// TIA Portal V21 program export: 7 tag tables, 1 data types, 2 data blocks, 11 code blocks (in call order from the OBs), 0 instance data blocks

VAR_GLOBAL   // PLC tag table "INSTRUMENTOS_ALARMES (ETA)"
   "NIVEL_MUITO_ALTO (ETA)" AT %M60.0 : Bool;
   "PRESSAO_ALTA (ETA)" AT %M60.1 : Bool;
END_VAR

VAR_GLOBAL   // PLC tag table "INSTRUMENTOS (ETA)"
   "FIT-01_STS" AT %M61.0 : Bool;
   "LIT-01_STS" AT %M61.1 : Bool;
END_VAR

VAR_GLOBAL   // PLC tag table "LadderTags"
   Start AT %M26.0 : Bool;
   Stop AT %M26.1 : Bool;
   Cmd_Motor1 AT %M26.2 : Bool;
   Falha_M1 AT %M26.3 : Bool;
   Nivel_Alto AT %M26.4 : Bool;
   Auto AT %M26.5 : Bool;
   Alarme AT %M26.6 : Bool;
   Reset AT %M26.7 : Bool;
   Manutencao AT %M27.0 : Bool;
   Pronto AT %M27.1 : Bool;
   Sensor_Falha AT %M27.2 : Bool;
   Temp_OK AT %M27.3 : Bool;
   Temperatura AT %MW28 : Int;
   Setpoint AT %MW30 : Int;
END_VAR

VAR_GLOBAL   // PLC tag table "SmokeTags"
   Smoke_Bit AT %M10.0 : Bool;
   Smoke_Out AT %M10.1 : Bool;
   Smoke_Int AT %MW12 : Int;
END_VAR

VAR_GLOBAL   // PLC tag table "PARTIDAS (ETA)"
   "ETA-P01_FALHA" AT %M60.2 : Bool;
END_VAR

VAR_GLOBAL   // PLC tag table "SOPRADOR_DESARENADOR (S-01A)"
   "S-01A_RESERVA_01" AT %M5512.0 : Bool;
   "S-01A_RESERVA_02" AT %M5512.1 : Bool;
   "S-01A_RESERVA_DINT_01" AT %MD5513 : DInt;
   "S-01A_STS_HABILITA_IMPAR_&" AT %M5506.4 : Bool;   // Status: Condições para partida do equipamento S-01A estão OK
   "S-01A_FALHA" AT %M5500.7 : Bool;   // Status: Falha geral do equipamento S-01A
   "S-01A_STS_FALHA_NAO_LIGOU" AT %M5506.1 : Bool;   // Status: Falha de partida do equipamento S-01A
   "S-01A_CMD_HABILITA_LIGA_AUTO2" AT %M5500.2 : Bool;   // Comando: Habilitação para partida em modo automático para o equipamento S-01A
   "S-01A_SP_SETPOINT_AUTO" AT %MW5502 : Int;   // Setpoint: Valor de referência em modo automático para o equipamento S-01A
   "S-01A_STS_HABILITA_PAR_&" AT %M5506.5 : Bool;   // Status: Condições para partida do equipamento S-01A estão OK
   "S-01A_CMD_BOTAO_RESET_FALHA" AT %M5500.0 : Bool;   // Comando: Botão de reset de falhas para o equipamento S-01A
   "S-01A_STS_VAR_MONITORADA" AT %MD5508 : Real;   // Status: Variável monitorada (Ex: vibração, temperatura) do equipamento S-01A
   "S-01A_STS_REMOTO_AUTO" AT %M5507.3 : Bool;   // Status: Comando Remoto em modo Automático para o equipamento S-01A
   "S-01A_STS_REMOTO_MANUAL" AT %M5507.4 : Bool;   // Status: Comando Remoto em modo Manual para o equipamento S-01A
   "S-01A_STS_LIGADO_PROFINET" AT %M5506.6 : Bool;   // Status: Comunicação Profinet OK com o equipamento S-01A
   "S-01A_STS_ALTERNANCIA_OK" AT %M5506.0 : Bool;   // Tag de controle/status/falha para o equipamento S-01A
   "S-01A_CMD_RESET_LIGA" AT %M5500.6 : Bool;   // Comando: Reset do comando Ligar o equipamento S-01A
   "S-01A_CMD_RESET_FALHA_PROFINET" AT %M5500.5 : Bool;   // Comando: Reset de falha Profinet para o equipamento S-01A
   "S-01A_STS_MODO_REMOTO" AT %M5507.2 : Bool;   // Status: Chave seletora do equipamento S-01A em Remoto
   "S-01A_LIGADO" AT %M5501.0 : Bool;   // Status: Equipamento S-01A em operação
   "S-01A_CMD_HABILITA_LIGA_AUTO" AT %M5500.1 : Bool;   // Comando: Habilitação para partida em modo automático para o equipamento S-01A
   "S-01A_STS_LOCAL_MANUAL" AT %M5507.0 : Bool;   // Status: Comando Local em modo Manual para o equipamento S-01A
   "S-01A_STS_FALHA_PROFINET" AT %M5506.2 : Bool;   // Status: Falha de comunicação Profinet com o equipamento S-01A
   "S-01A_STS_SUCCAO_OK" AT %M5507.5 : Bool;   // Status: Condição de sucção OK para a bomba S-01A
   "S-01A_STS_MODO_LOCAL" AT %M5507.1 : Bool;   // Status: Chave seletora do equipamento S-01A em Local
   "S-01A_STS_HABILITA" AT %M5506.3 : Bool;   // Status: Condições para partida do equipamento S-01A estão OK
   "S-01A_STS_LOCAL_AUTO" AT %M5506.7 : Bool;   // Status: Comando Local em modo Automático para o equipamento S-01A
   "S-01A_CMD_LIGA_PROFINET" AT %M5500.4 : Bool;   // Comando: Partida via Profinet para o equipamento S-01A
   "S-01A_SP_SETPOINT_MANUAL" AT %MW5504 : Int;   // Setpoint: Valor de referência em modo manual para o equipamento S-01A
   "S-01A_CMD_LIGA_BOMBA" AT %M5500.3 : Bool;   // Comando: Ligar/Partir a bomba S-01A
END_VAR

VAR_GLOBAL   // PLC tag table "BOMBA (BH-01B)"
END_VAR

TYPE "MotorDados"
VERSION : 0.1
   STRUCT
      Liga : Bool;
      Ligado : Bool;
      Numero : Int;
   END_STRUCT;
END_TYPE

DATA_BLOCK "DB GLOBAL"
{ S7_Optimized_Access := 'TRUE' }
VERSION : 0.1
   STRUCT
      "Motor_BH-01A" : "MotorDados";
      "Motor_BH-01B" : "MotorDados";
   END_STRUCT;

BEGIN
END_DATA_BLOCK

DATA_BLOCK "ALARMES_MODULOS"
{ S7_Optimized_Access := 'TRUE' }
VERSION : 0.1
   STRUCT
      "QA-01" : STRUCT
         WORD_1 : Word;
         WORD_2 : Word;
      END_STRUCT;
   END_STRUCT;

BEGIN
END_DATA_BLOCK

DATA_BLOCK "DB INSTRUMENTOS"
{ S7_Optimized_Access := 'TRUE' }
VERSION : 0.1
   STRUCT
      ETA : STRUCT
         "FIT-01" : STRUCT
            WORD_STS : Word;
            CMD_AF : Int;
            CMD_LIM : Int;
         END_STRUCT;
         "LIT-01" : STRUCT
            WORD_STS : Word;
            CMD_AF : Int;
            CMD_LIM : Int;
         END_STRUCT;
      END_STRUCT;
   END_STRUCT;

BEGIN
END_DATA_BLOCK

DATA_BLOCK "DB_BITS_TO_WORD_FIT-01"
{ S7_Optimized_Access := 'TRUE' }
VERSION : 0.1
"FB BITS TO WORD"

BEGIN
END_DATA_BLOCK

ORGANIZATION_BLOCK "OB_MOLDE_ALARMES"   // OB1, LAD, ProgramCycle
TITLE = "Main Program Sweep (Cycle)"
{ S7_Optimized_Access := 'TRUE' }
VERSION : 0.1
// stored: AutoNumber true, IsIECCheckEnabled false, SetENOAutomatically false
   VAR_INPUT
      Initial_Call : Bool;   // Initial call of this OB
      Remanence : Bool;   // =True, if remanent data are available
   END_VAR
BEGIN

REGION Network 1: FC Alarmes: Paineis
   // comentário da chamada da fc 1
END_REGION
END_ORGANIZATION_BLOCK

ORGANIZATION_BLOCK "MODULE_ERROR_MOLDE"   // OB123, LAD, ProgramCycle
TITLE = MODULE_ERROR_MOLDE
{ S7_Optimized_Access := 'TRUE' }
VERSION : 0.1
// stored: AutoNumber true, IsIECCheckEnabled false, SetENOAutomatically false
   VAR_INPUT
      Initial_Call : Bool;
      Remanence : Bool;
   END_VAR
BEGIN

REGION Network 1: Molde: falha modulo HW 999
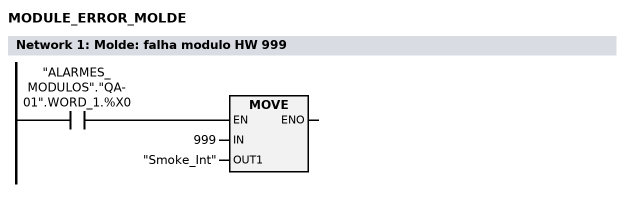
   RUNG wire#powerrail
      Contact( "ALARMES_MODULOS"."QA-01".WORD_1.%X0 )
      { S7_GenerateENO := "TRUE" } Move(in := 999, out1 := "Smoke_Int")
   END_RUNG
   // the same network as SCL:
   IF "ALARMES_MODULOS"."QA-01".WORD_1.%X0 THEN <??.?> := 999; END_IF;
END_REGION
END_ORGANIZATION_BLOCK

ORGANIZATION_BLOCK "OB_INSTRUMENTOS"   // OB130, LAD, ProgramCycle
TITLE = OB_INSTRUMENTOS
{ S7_Optimized_Access := 'TRUE' }
VERSION : 0.1
// stored: AutoNumber true, IsIECCheckEnabled false, SetENOAutomatically false
   VAR_INPUT
      Initial_Call : Bool;
      Remanence : Bool;
   END_VAR
BEGIN
END_ORGANIZATION_BLOCK

FUNCTION "PARTIDA_SOPRADOR_1 (S-01A)" : Void   // FC148, LAD
{ S7_Optimized_Access := 'TRUE' }
VERSION : 0.1
// Network 1: Set memórias entradas digitais
// Network 2: Function Block FALHA
// Network 3: MODO AUTOMÁTICO: Condições para Modo Automático
// Network 4: Alternância/Rotatividade de bombas Principal-Reserva
// Network 5: Function Block CONDIÇÃO DE PARTIDA
// Network 6: Setpoint Manual - Velocidade Proporcial ao Sinal de Saída
// Network 7: Reset Comando Liga
// Network 8: Intertravamento para habilitar o botão liga na IHM
// Network 9: Intertravamento de Segurança
// Network 10: Bloco de Controle Inversor Profinet
// Network 11: Aciona saída digital para partir o motor/bomba
// Network 1: Set memórias entradas digitais
// Network 2: Function Block FALHA
// Network 3: MODO AUTOMÁTICO: Condições para Modo Automático
// Network 4: Alternância/Rotatividade de bombas Principal-Reserva
// Network 5: Function Block CONDIÇÃO DE PARTIDA
// Network 6: Reset Comando Liga
// Network 7: Function Block MODOS DE OPERAÇÃO - Atribuição dos Modos de Operação
// Network 8: Intertravamento para habilitar o botão liga na IHM
// Network 9: Intertravamento de Segurança
// Network 10: Function Block SUCÇÃO OK
// Network 11: Aciona saída digital para partir o motor/bomba
// Network 12: Function Block HORÍMETRO - Tempo de bomba ligada em horas
// stored: AutoNumber true, IsIECCheckEnabled false, SetENOAutomatically false, UDAEnableTagReadback false
   VAR_TEMP   // added for the SCL form of the ladder/FBD networks
      _w1 : Bool;
   END_VAR
BEGIN

REGION Network 1: Set memórias entradas digitais
   // Instanciando entradas digitais em PLC Tags "%M " Address
   // 
   // MODO LOCAL: Indica Operação Local da bomba.
   // MODO REMOTO: Indica Operação Remoto da bomba (IHM).
   // LIGADO: Indica bomba ligada (caso, via sinal discreto).
   // FALHA: Sinal de Falha (caso, via sinal discreto).
   // Instanciando entradas digitais em PLC Tags "M" Address
   // 
   // MODO LOCAL: Indica Operação Local da bomba
   // MODO REMOTO: Indica Operação Remoto da bomba (IHM)
   // LIGADO: Indica bomba ligada
   // FALHA: Sinal de Falha
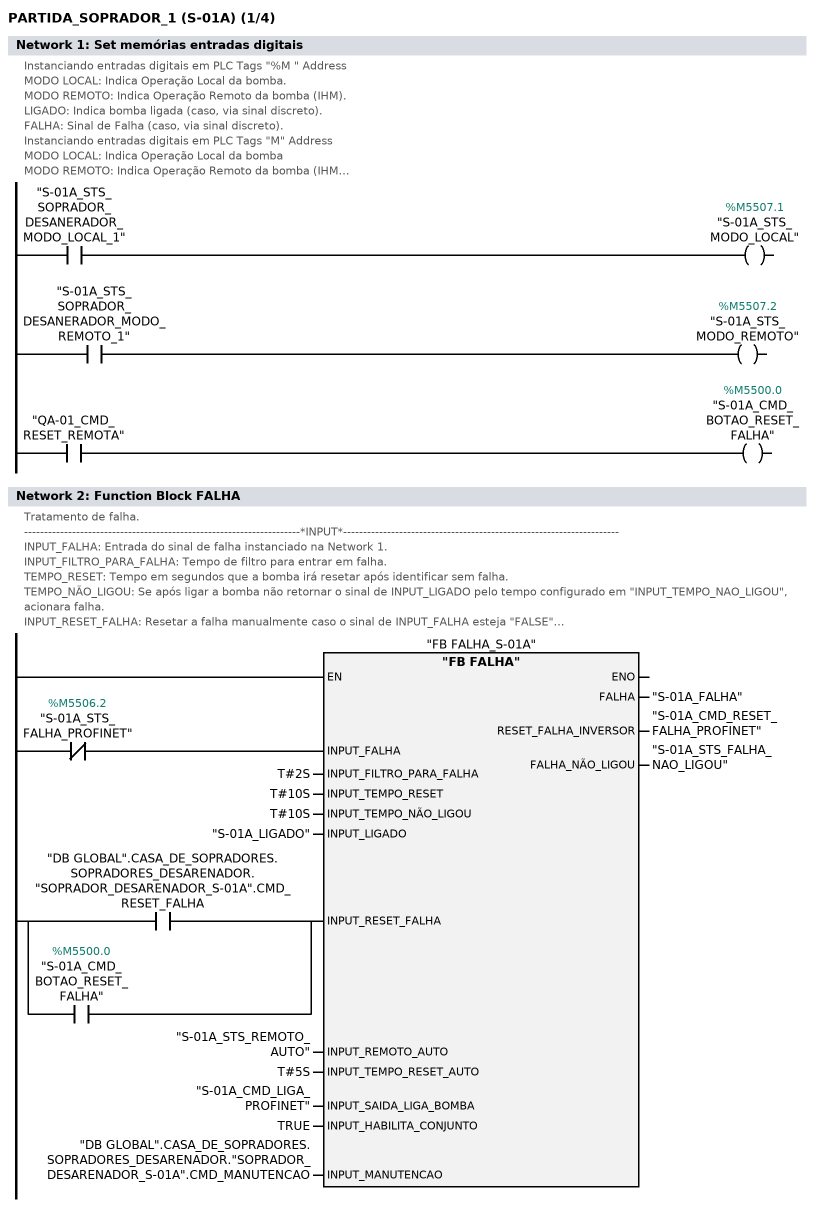
   RUNG wire#powerrail
      Contact( "S-01A_STS_SOPRADOR_DESANERADOR_MODO_LOCAL_1" )
      Coil( "S-01A_STS_MODO_LOCAL" )
   END_RUNG
   RUNG wire#powerrail
      Contact( "S-01A_STS_SOPRADOR_DESANERADOR_MODO_REMOTO_1" )
      Coil( "S-01A_STS_MODO_REMOTO" )
   END_RUNG
   RUNG wire#powerrail
      Contact( "QA-01_CMD_RESET_REMOTA" )
      Coil( "S-01A_CMD_BOTAO_RESET_FALHA" )
   END_RUNG
   // the same network as SCL:
   "S-01A_STS_MODO_LOCAL" := "S-01A_STS_SOPRADOR_DESANERADOR_MODO_LOCAL_1";
   "S-01A_STS_MODO_REMOTO" := "S-01A_STS_SOPRADOR_DESANERADOR_MODO_REMOTO_1";
   "S-01A_CMD_BOTAO_RESET_FALHA" := "QA-01_CMD_RESET_REMOTA";
END_REGION

REGION Network 2: Function Block FALHA
   // Tratamento de falha.
   // ---------------------------------------------------------------------*INPUT*---------------------------------------------------------------------
   // INPUT_FALHA: Entrada do sinal de falha instanciado na Network 1.
   // INPUT_FILTRO_PARA_FALHA: Tempo de filtro para entrar em falha.
   // TEMPO_RESET: Tempo em segundos que a bomba irá resetar após identificar sem falha.
   // TEMPO_NÃO_LIGOU: Se após ligar a bomba não retornar o sinal de INPUT_LIGADO pelo tempo configurado em "INPUT_TEMPO_NAO_LIGOU", acionara falha.
   // INPUT_RESET_FALHA: Resetar a falha manualmente caso o sinal de INPUT_FALHA esteja "FALSE".
   // INPUT_REMOTO_AUTO: Caso o equipamento entrar em estado de "FALHA" em "REMOTO_AUTOMATICO" o bloco fará um reset com atraso pelo tempo "INPUT_TEMPO_RESET_AUTO".
   // INPUT_TEMPO_RESET_AUTO: Caso em "REMOTO_AUTO", para resetar será contado o tempo de entrada.
   // INPUT_SAIDA_LIGA_BOMBA: Comando de saída para acionar o equipamento.
   // INPUT_HABILITA_CONJUNTO: Comando para casos de Principal e Reserva (padrão "TRUE").
   // INPUT_MANUTENCAO: Comando de manutenção do equipamento intertrava qualquer acionamento e status de "FALHA".
   // ---------------------------------------------------------------------*OUTPUT*---------------------------------------------------------------------
   // FALHA: Sinal de saída de "FALHA" do equipamento.
   // RESET_FALHA_INVERSOR: Comando enviado para reset do inversor em caso de "FALHA".
   // FALHA_NAO_LIGOU: Caso esteja sendo enviado o comando para "LIGAR" e não receber o feedback de ligado, no tempo de "TEMPO_NÃO_LIGOU", o equiapamento entra em "FALHA".
   // Tratamento de falha da bomba
   // INPUT_FALHA: Entrada do sinal de falha instanciado na Network 1.
   // TEMPO_RESET: Tempo em segundos que a bomba irá resetar após identificar sem falha.
   // TEMPO_NÃO_LIGOU: Se após ligar a bomba não retornar o sinal de LIGADO pelo tempo configurado, acionara falha.
   // INPUT_RESET_FALHA: Resetar a falha manualmente caso o sinal de INPUT_FALHA esteja FALSE
   RUNG wire#powerrail
      "FB FALHA_S-01A"(INPUT_FALHA := wire#w1, INPUT_RESET_FALHA := wire#w2, INPUT_FILTRO_PARA_FALHA := T#2S, INPUT_TEMPO_RESET := T#10S, INPUT_TEMPO_NÃO_LIGOU := T#10S, INPUT_LIGADO := "S-01A_LIGADO", INPUT_REMOTO_AUTO := "S-01A_STS_REMOTO_AUTO", INPUT_TEMPO_RESET_AUTO := T#5S, INPUT_SAIDA_LIGA_BOMBA := "S-01A_CMD_LIGA_PROFINET", INPUT_HABILITA_CONJUNTO := TRUE, INPUT_MANUTENCAO := "DB GLOBAL".CASA_DE_SOPRADORES.SOPRADORES_DESARENADOR."SOPRADOR_DESARENADOR_S-01A".CMD_MANUTENCAO, FALHA => "S-01A_FALHA", RESET_FALHA_INVERSOR => "S-01A_CMD_RESET_FALHA_PROFINET", FALHA_NÃO_LIGOU => "S-01A_STS_FALHA_NAO_LIGOU")
   END_RUNG
   RUNG wire#powerrail
      I_Contact( "S-01A_STS_FALHA_PROFINET" )
   END_RUNG wire#w1
   RUNG wire#powerrail
      Contact( "DB GLOBAL".CASA_DE_SOPRADORES.SOPRADORES_DESARENADOR."SOPRADOR_DESARENADOR_S-01A".CMD_RESET_FALHA )
   END_RUNG wire#w2
   RUNG wire#powerrail
      Contact( "S-01A_CMD_BOTAO_RESET_FALHA" )
   END_RUNG wire#w2
   // the same network as SCL:
   "FB FALHA_S-01A"(INPUT_FALHA := NOT "S-01A_STS_FALHA_PROFINET",   // "FB FALHA"
                    INPUT_FILTRO_PARA_FALHA := T#2S,
                    INPUT_TEMPO_RESET := T#10S,
                    INPUT_TEMPO_NÃO_LIGOU := T#10S,
                    INPUT_LIGADO := "S-01A_LIGADO",
                    INPUT_RESET_FALHA := "DB GLOBAL".CASA_DE_SOPRADORES.SOPRADORES_DESARENADOR."SOPRADOR_DESARENADOR_S-01A".CMD_RESET_FALHA OR "S-01A_CMD_BOTAO_RESET_FALHA",
                    INPUT_REMOTO_AUTO := "S-01A_STS_REMOTO_AUTO",
                    INPUT_TEMPO_RESET_AUTO := T#5S,
                    INPUT_SAIDA_LIGA_BOMBA := "S-01A_CMD_LIGA_PROFINET",
                    INPUT_HABILITA_CONJUNTO := TRUE,
                    INPUT_MANUTENCAO := "DB GLOBAL".CASA_DE_SOPRADORES.SOPRADORES_DESARENADOR."SOPRADOR_DESARENADOR_S-01A".CMD_MANUTENCAO,
                    FALHA => "S-01A_FALHA",
                    RESET_FALHA_INVERSOR => "S-01A_CMD_RESET_FALHA_PROFINET",
                    FALHA_NÃO_LIGOU => "S-01A_STS_FALHA_NAO_LIGOU");
END_REGION

REGION Network 3: MODO AUTOMÁTICO: Condições para Modo Automático
   // ----------------------------------------------------------------------*INPUT*---------------------------------------------------------------------
   // ---------------------------------------------------------------------*OUTPUT*------------------------------------------------------------------
END_REGION

REGION Network 4: Alternância/Rotatividade de bombas Principal-Reserva
   // ----------------------------------------------------------------------*INPUT*---------------------------------------------------------------------
   // ---------------------------------------------------------------------*OUTPUT*------------------------------------------------------------------
END_REGION

REGION Network 5: Function Block CONDIÇÃO DE PARTIDA
   // Varredura de condicionais para ligar
   // ----------------------------------------------------------------------*INPUT*---------------------------------------------------------------------
   // INPUT_LIGADO: Entrada do sinal de ligado instanciado na Network 1.
   // INPUT_DESLIGADO: Entrada do sinal discreto "DESLIGADO" (caso, feedback via sinal discreto).
   // INPUT_FALHA: Entrada do sinal de falha da saída do bloco na Network 2.
   // INPUT_LOCAL: Entrada do sinal de modo local instanciado na Network 1.
   // INPUT_LOC_AUTO: Entrada do sinal do modo Local Automático
   // INPUT_REMOTO: Entrada do sinal de modo remoto instanciado na Network 1.
   // INPUT_FALHA_PROFNET: Entrada do sinal de Falha na comunicação Profinet.
   // INPUT_HABILITA_AUTO: Entrada do Sinal que habilita o modo Automático.
   // INPUT_CMD_LIGA: Entrada do sinal para acionar o equipamento.
   // CMD_MANUTENÇÃO:Comando de manutenção do equipamento intertrava qualquer acionamento.
   // CMD_MODO_OPERAÇÃO: Seleção do modo de operação do equipamento.
   // CMD_RESET_HORIMETRO: Comando para resetar o contador de Horas Trabalhadas.
   // 
   // 
   // ---------------------------------------------------------------------*OUTPUT*------------------------------------------------------------------
   // LIGA_BOMBA: Se TRUE, as condições estão OK para ligar na Network 11.
   // STATUS_MOTOR: Status de saída; 0 = DESLIGADO; 1 = LIGADO; 2 = FALHA; 3 = MANUTENÇÃO.
   // OUTPUT_REMOTO_AUTO: Saída indica que o motor/bomba está em modo Remoto Automático.
   // OUTPUT_MODO_OPERAÇÃO: Modo de operação local/remoto, manual/automático do equipamento
   // STS_HORIMETRO: Contabilização do tempo do equipamento em operação.
   // RESET_CMD_LIGA: Reset da memória de comando "LIGA" em casos do equipamento estar em modo "REMOTO_AUTOMATICO" ou "FALHA" ou "MANUTENÇÃO".
   // Varredura de condicionais para ligar
   // INPUT_LIGADO: Entrada do sinal de ligado instanciado na Network 1.
   // INPUT_FALHA: Entrada do sinal de falha da saída do bloco na Network 2.
   // INPUT_LOCAL: Entrada do sinal de modo local instanciado na Network 1.
   // INPUT_LOC_AUTO: Entrada do sinal do modo Local Automático
   // INPUT_REMOTO: Entrada do sinal de modo remoto instanciado na Network 1.
   // PARÂMETRO: Parâmetro de monitoramento para ligar e desligar a bomba em automático.
   // PARÂMETRO_LIGA/DESLIGA: Cadastros de programação liga/desliga em relação ao parâmetro.
   // CMD: Comandos recebidos pelo bloco
   // STATUS_MOTOR: Status de saída; 0 = DESLIGADO; 1 = LIGADO; 2 = FALHA; 3 = MANUTENÇÃO.
   // LIGA_BOMBA: Se TRUE, as condições estão OK para ligar na 5.
   // REMOTO_MAN: Saída indica que o motor/bomba está em modo Remoto Manual
   // REMOTO_AUTO: Saída indica que o motor/bomba está em modo Remoto Automático
   // LOCAL_MAN: Saída indica que o motor/bomba está em modo Local Manual
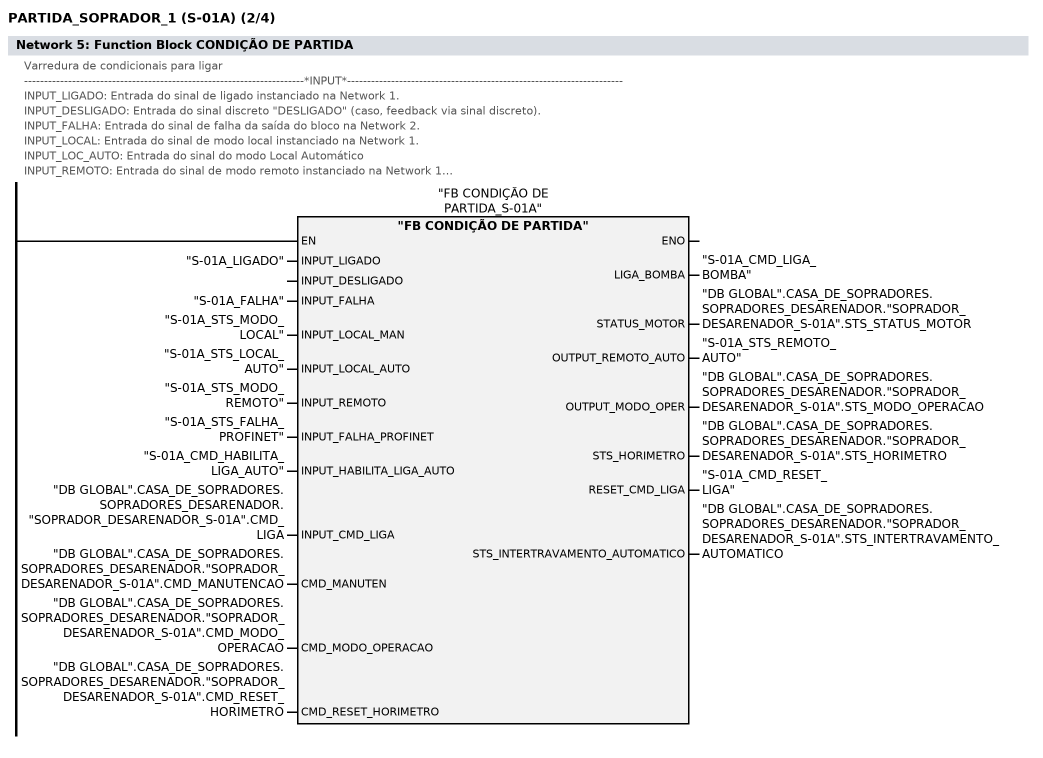
   RUNG wire#powerrail
      "FB CONDIÇÃO DE PARTIDA_S-01A"(INPUT_LIGADO := "S-01A_LIGADO", INPUT_DESLIGADO :=, INPUT_FALHA := "S-01A_FALHA", INPUT_LOCAL_MAN := "S-01A_STS_MODO_LOCAL", INPUT_LOCAL_AUTO := "S-01A_STS_LOCAL_AUTO", INPUT_REMOTO := "S-01A_STS_MODO_REMOTO", INPUT_FALHA_PROFINET := "S-01A_STS_FALHA_PROFINET", INPUT_HABILITA_LIGA_AUTO := "S-01A_CMD_HABILITA_LIGA_AUTO", INPUT_CMD_LIGA := "DB GLOBAL".CASA_DE_SOPRADORES.SOPRADORES_DESARENADOR."SOPRADOR_DESARENADOR_S-01A".CMD_LIGA, CMD_MANUTEN := "DB GLOBAL".CASA_DE_SOPRADORES.SOPRADORES_DESARENADOR."SOPRADOR_DESARENADOR_S-01A".CMD_MANUTENCAO, CMD_MODO_OPERACAO := "DB GLOBAL".CASA_DE_SOPRADORES.SOPRADORES_DESARENADOR."SOPRADOR_DESARENADOR_S-01A".CMD_MODO_OPERACAO, CMD_RESET_HORIMETRO := "DB GLOBAL".CASA_DE_SOPRADORES.SOPRADORES_DESARENADOR."SOPRADOR_DESARENADOR_S-01A".CMD_RESET_HORIMETRO, LIGA_BOMBA => "S-01A_CMD_LIGA_BOMBA", STATUS_MOTOR => "DB GLOBAL".CASA_DE_SOPRADORES.SOPRADORES_DESARENADOR."SOPRADOR_DESARENADOR_S-01A".STS_STATUS_MOTOR, OUTPUT_REMOTO_AUTO => "S-01A_STS_REMOTO_AUTO", OUTPUT_MODO_OPER => "DB GLOBAL".CASA_DE_SOPRADORES.SOPRADORES_DESARENADOR."SOPRADOR_DESARENADOR_S-01A".STS_MODO_OPERACAO, STS_HORIMETRO => "DB GLOBAL".CASA_DE_SOPRADORES.SOPRADORES_DESARENADOR."SOPRADOR_DESARENADOR_S-01A".STS_HORIMETRO, RESET_CMD_LIGA => "S-01A_CMD_RESET_LIGA", STS_INTERTRAVAMENTO_AUTOMATICO => "DB GLOBAL".CASA_DE_SOPRADORES.SOPRADORES_DESARENADOR."SOPRADOR_DESARENADOR_S-01A".STS_INTERTRAVAMENTO_AUTOMATICO)
   END_RUNG
   // the same network as SCL:
   "FB CONDIÇÃO DE PARTIDA_S-01A"(INPUT_LIGADO := "S-01A_LIGADO",   // "FB CONDIÇÃO DE PARTIDA"
                           INPUT_FALHA := "S-01A_FALHA",
                           INPUT_LOCAL_MAN := "S-01A_STS_MODO_LOCAL",
                           INPUT_LOCAL_AUTO := "S-01A_STS_LOCAL_AUTO",
                           INPUT_REMOTO := "S-01A_STS_MODO_REMOTO",
                           INPUT_FALHA_PROFINET := "S-01A_STS_FALHA_PROFINET",
                           INPUT_HABILITA_LIGA_AUTO := "S-01A_CMD_HABILITA_LIGA_AUTO",
                           INPUT_CMD_LIGA := "DB GLOBAL".CASA_DE_SOPRADORES.SOPRADORES_DESARENADOR."SOPRADOR_DESARENADOR_S-01A".CMD_LIGA,
                           CMD_MANUTEN := "DB GLOBAL".CASA_DE_SOPRADORES.SOPRADORES_DESARENADOR."SOPRADOR_DESARENADOR_S-01A".CMD_MANUTENCAO,
                           CMD_MODO_OPERACAO := "DB GLOBAL".CASA_DE_SOPRADORES.SOPRADORES_DESARENADOR."SOPRADOR_DESARENADOR_S-01A".CMD_MODO_OPERACAO,
                           CMD_RESET_HORIMETRO := "DB GLOBAL".CASA_DE_SOPRADORES.SOPRADORES_DESARENADOR."SOPRADOR_DESARENADOR_S-01A".CMD_RESET_HORIMETRO,
                           LIGA_BOMBA => "S-01A_CMD_LIGA_BOMBA",
                           STATUS_MOTOR => "DB GLOBAL".CASA_DE_SOPRADORES.SOPRADORES_DESARENADOR."SOPRADOR_DESARENADOR_S-01A".STS_STATUS_MOTOR,
                           OUTPUT_REMOTO_AUTO => "S-01A_STS_REMOTO_AUTO",
                           OUTPUT_MODO_OPER => "DB GLOBAL".CASA_DE_SOPRADORES.SOPRADORES_DESARENADOR."SOPRADOR_DESARENADOR_S-01A".STS_MODO_OPERACAO,
                           STS_HORIMETRO => "DB GLOBAL".CASA_DE_SOPRADORES.SOPRADORES_DESARENADOR."SOPRADOR_DESARENADOR_S-01A".STS_HORIMETRO,
                           RESET_CMD_LIGA => "S-01A_CMD_RESET_LIGA",
                           STS_INTERTRAVAMENTO_AUTOMATICO => "DB GLOBAL".CASA_DE_SOPRADORES.SOPRADORES_DESARENADOR."SOPRADOR_DESARENADOR_S-01A".STS_INTERTRAVAMENTO_AUTOMATICO);
END_REGION

REGION Network 6: Setpoint Manual - Velocidade Proporcial ao Sinal de Saída
   // Function Block SETPOINT UNIT TO RPM = Recebe o setpoint da IHM em L/h e o converte em RPM
   // ----------------------------------------------------------------------*INPUT*---------------------------------------------------------------------
   // MAX_RPM = Valor cadastrado para definir qual o valor que corresponde ao RPM máximo
   // MIN_RPM = Valor cadastrado para definir qual o valor que corresponde àao RPM mínimo
   // SETPOINT = Valor recebido em L/h
   // 
   // Function Block SETPOINT_MANUAL = Recebe o setpoint convertido em RPM e calcula a referência de velocidade proporcional baseando-se no fundo de escala
   // REMOTO_COMANDO_VALOR = Valor de comando para comparação
   // COMANDO = Comando recebido para confirmar setpoint
   // RANGE_MAX: Valor cadastrado para definir qual o valor que corresponde ao RPM máximo
   // RANGE_MIN: Valor cadastrado para definir qual o valor que corresponde àao RPM mínimo
   // VALOR_SAIDA: Valor do setpoint interpretado dentro da escala do CLP correspondente ao sinal elétrico (4-20mA ou 0-10V) que o inversor recebe e ajusta sua saída proporcionalmente.
   // 
   // ---------------------------------------------------------------------*OUTPUT*------------------------------------------------------------------
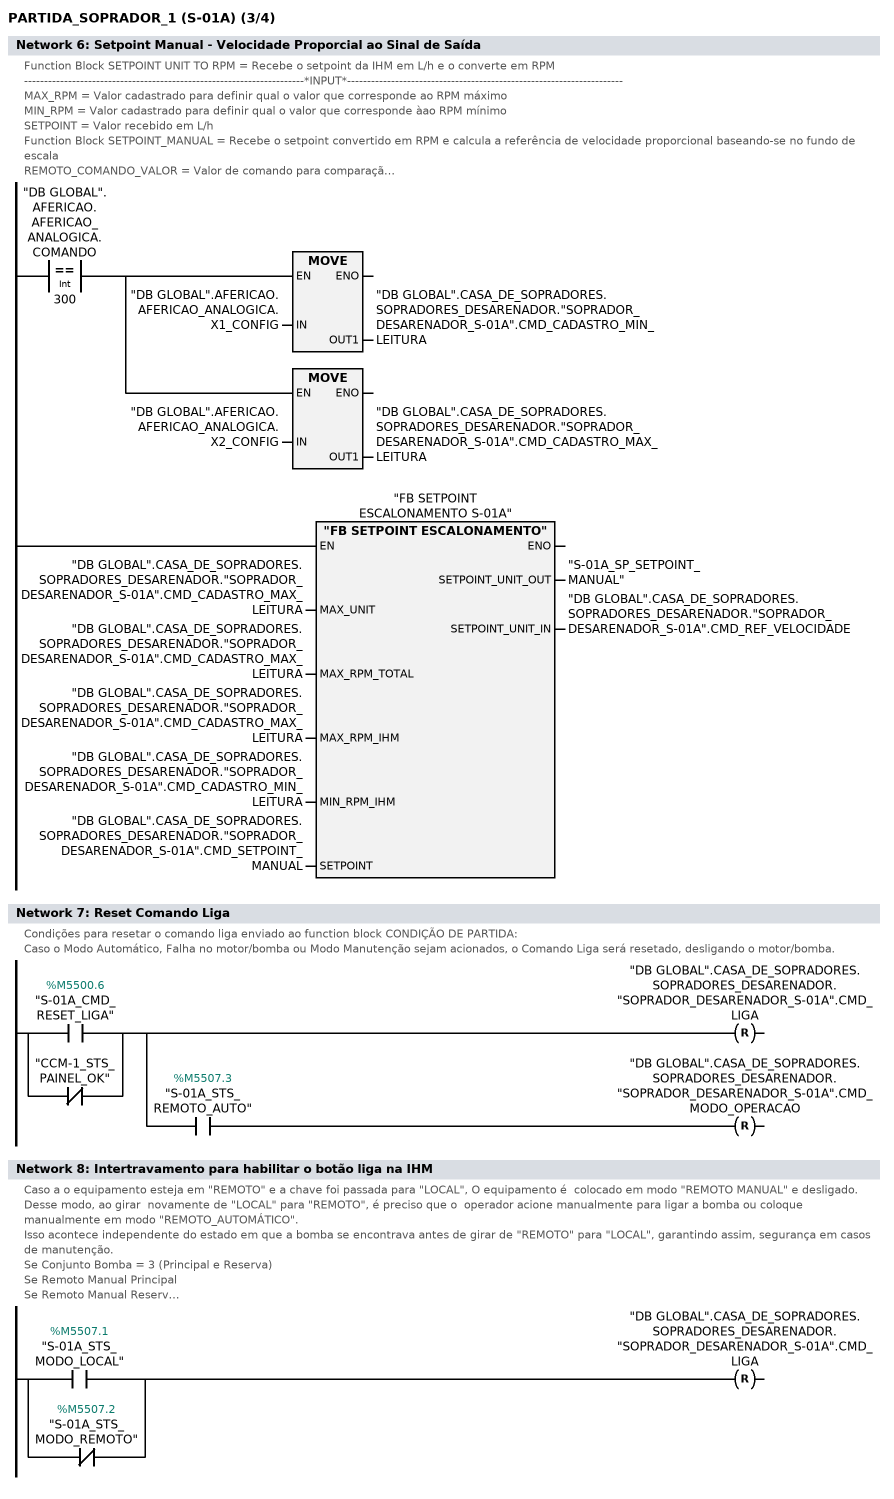
   RUNG wire#powerrail
      { S7_Templates := "SrcType := Int" } EQ_Contact(in1 := "DB GLOBAL".AFERICAO.AFERICAO_ANALOGICA.COMANDO, in2 := 300)
      wire#w1
      Move(in := "DB GLOBAL".AFERICAO.AFERICAO_ANALOGICA.X1_CONFIG, out1 => "DB GLOBAL".CASA_DE_SOPRADORES.SOPRADORES_DESARENADOR."SOPRADOR_DESARENADOR_S-01A".CMD_CADASTRO_MIN_LEITURA)
   END_RUNG
   RUNG wire#w1
      Move(in := "DB GLOBAL".AFERICAO.AFERICAO_ANALOGICA.X2_CONFIG, out1 => "DB GLOBAL".CASA_DE_SOPRADORES.SOPRADORES_DESARENADOR."SOPRADOR_DESARENADOR_S-01A".CMD_CADASTRO_MAX_LEITURA)
   END_RUNG
   RUNG wire#powerrail
      "FB SETPOINT ESCALONAMENTO S-01A"(MAX_UNIT := "DB GLOBAL".CASA_DE_SOPRADORES.SOPRADORES_DESARENADOR."SOPRADOR_DESARENADOR_S-01A".CMD_CADASTRO_MAX_LEITURA, MAX_RPM_TOTAL := "DB GLOBAL".CASA_DE_SOPRADORES.SOPRADORES_DESARENADOR."SOPRADOR_DESARENADOR_S-01A".CMD_CADASTRO_MAX_LEITURA, MAX_RPM_IHM := "DB GLOBAL".CASA_DE_SOPRADORES.SOPRADORES_DESARENADOR."SOPRADOR_DESARENADOR_S-01A".CMD_CADASTRO_MAX_LEITURA, MIN_RPM_IHM := "DB GLOBAL".CASA_DE_SOPRADORES.SOPRADORES_DESARENADOR."SOPRADOR_DESARENADOR_S-01A".CMD_CADASTRO_MIN_LEITURA, SETPOINT := "DB GLOBAL".CASA_DE_SOPRADORES.SOPRADORES_DESARENADOR."SOPRADOR_DESARENADOR_S-01A".CMD_SETPOINT_MANUAL, SETPOINT_UNIT_OUT => "S-01A_SP_SETPOINT_MANUAL", SETPOINT_UNIT_IN => "DB GLOBAL".CASA_DE_SOPRADORES.SOPRADORES_DESARENADOR."SOPRADOR_DESARENADOR_S-01A".CMD_REF_VELOCIDADE)
   END_RUNG
   // the same network as SCL:
   IF "DB GLOBAL".AFERICAO.AFERICAO_ANALOGICA.COMANDO = 300 THEN
       "DB GLOBAL".CASA_DE_SOPRADORES.SOPRADORES_DESARENADOR."SOPRADOR_DESARENADOR_S-01A".CMD_CADASTRO_MIN_LEITURA := "DB GLOBAL".AFERICAO.AFERICAO_ANALOGICA.X1_CONFIG;
       "DB GLOBAL".CASA_DE_SOPRADORES.SOPRADORES_DESARENADOR."SOPRADOR_DESARENADOR_S-01A".CMD_CADASTRO_MAX_LEITURA := "DB GLOBAL".AFERICAO.AFERICAO_ANALOGICA.X2_CONFIG;
   END_IF;
   "FB SETPOINT ESCALONAMENTO S-01A"(MAX_UNIT := "DB GLOBAL".CASA_DE_SOPRADORES.SOPRADORES_DESARENADOR."SOPRADOR_DESARENADOR_S-01A".CMD_CADASTRO_MAX_LEITURA,   // "FB SETPOINT ESCALONAMENTO"
                           MAX_RPM_TOTAL := "DB GLOBAL".CASA_DE_SOPRADORES.SOPRADORES_DESARENADOR."SOPRADOR_DESARENADOR_S-01A".CMD_CADASTRO_MAX_LEITURA,
                           MAX_RPM_IHM := "DB GLOBAL".CASA_DE_SOPRADORES.SOPRADORES_DESARENADOR."SOPRADOR_DESARENADOR_S-01A".CMD_CADASTRO_MAX_LEITURA,
                           MIN_RPM_IHM := "DB GLOBAL".CASA_DE_SOPRADORES.SOPRADORES_DESARENADOR."SOPRADOR_DESARENADOR_S-01A".CMD_CADASTRO_MIN_LEITURA,
                           SETPOINT := "DB GLOBAL".CASA_DE_SOPRADORES.SOPRADORES_DESARENADOR."SOPRADOR_DESARENADOR_S-01A".CMD_SETPOINT_MANUAL,
                           SETPOINT_UNIT_OUT => "S-01A_SP_SETPOINT_MANUAL",
                           SETPOINT_UNIT_IN => "DB GLOBAL".CASA_DE_SOPRADORES.SOPRADORES_DESARENADOR."SOPRADOR_DESARENADOR_S-01A".CMD_REF_VELOCIDADE);
END_REGION

REGION Network 7: Reset Comando Liga
   // Condições para resetar o comando liga enviado ao function block CONDIÇÃO DE PARTIDA:
   // Caso o Modo Automático, Falha no motor/bomba ou Modo Manutenção sejam acionados, o Comando Liga será resetado, desligando o motor/bomba.
   RUNG wire#powerrail
      Contact( "S-01A_CMD_RESET_LIGA" )
      wire#w1
      R_Coil( "DB GLOBAL".CASA_DE_SOPRADORES.SOPRADORES_DESARENADOR."SOPRADOR_DESARENADOR_S-01A".CMD_LIGA )
   END_RUNG
   RUNG wire#powerrail
      I_Contact( "CCM-1_STS_PAINEL_OK" )
   END_RUNG wire#w1
   RUNG wire#w1
      Contact( "S-01A_STS_REMOTO_AUTO" )
      R_Coil( "DB GLOBAL".CASA_DE_SOPRADORES.SOPRADORES_DESARENADOR."SOPRADOR_DESARENADOR_S-01A".CMD_MODO_OPERACAO )
   END_RUNG
   // the same network as SCL:
   #_w1 := "S-01A_CMD_RESET_LIGA" OR NOT "CCM-1_STS_PAINEL_OK";
   IF #_w1 THEN
       "DB GLOBAL".CASA_DE_SOPRADORES.SOPRADORES_DESARENADOR."SOPRADOR_DESARENADOR_S-01A".CMD_LIGA := FALSE;
   END_IF;
   IF #_w1 AND "S-01A_STS_REMOTO_AUTO" THEN
       "DB GLOBAL".CASA_DE_SOPRADORES.SOPRADORES_DESARENADOR."SOPRADOR_DESARENADOR_S-01A".CMD_MODO_OPERACAO := FALSE;
   END_IF;
END_REGION

REGION Network 8: Intertravamento para habilitar o botão liga na IHM
   // Caso a o equipamento esteja em "REMOTO" e a chave foi passada para "LOCAL", O equipamento é  colocado em modo "REMOTO MANUAL" e desligado.
   // Desse modo, ao girar  novamente de "LOCAL" para "REMOTO", é preciso que o  operador acione manualmente para ligar a bomba ou coloque manualmente em modo "REMOTO_AUTOMÁTICO".
   // Isso acontece independente do estado em que a bomba se encontrava antes de girar de "REMOTO" para "LOCAL", garantindo assim, segurança em casos de manutenção.
   // Se Conjunto Bomba = 3 (Principal e Reserva)
   // Se Remoto Manual Principal
   // Se Remoto Manual Reserva
   // Se Habilitado Liga Principal
   // Se Habilitado Liga Reserva
   // Então Habilita Conjunto de Bomba
   // 
   // Se Conjunto Bomba <> 3
   // Se Remoto Manual Principal
   // Se Habilita Principal 
   // ou
   // Se Remoto Manual Reserva 
   // Se Habilita Reserva
   // Então Habilita Bomba Unitária
   // 
   // Se Bomba Unitária Habilitado
   // ou
   // Se Conjunto Bomba Habilitado
   // Então 
   // Habilita Intertravamento Botão IHM de Conjunto Bomba
   RUNG wire#powerrail
      Contact( "S-01A_STS_MODO_LOCAL" )
      wire#w1
      R_Coil( "DB GLOBAL".CASA_DE_SOPRADORES.SOPRADORES_DESARENADOR."SOPRADOR_DESARENADOR_S-01A".CMD_LIGA )
   END_RUNG
   RUNG wire#powerrail
      I_Contact( "S-01A_STS_MODO_REMOTO" )
   END_RUNG wire#w1
   // the same network as SCL:
   IF "S-01A_STS_MODO_LOCAL" OR NOT "S-01A_STS_MODO_REMOTO" THEN
       "DB GLOBAL".CASA_DE_SOPRADORES.SOPRADORES_DESARENADOR."SOPRADOR_DESARENADOR_S-01A".CMD_LIGA := FALSE;
   END_IF;
END_REGION

REGION Network 9: Intertravamento de Segurança
   // Se {
   // Modo Local = False
   // e Se Local Automático = False
   // e Se Local Manual = False
   // e Se Modo Remoto = True
   // e Se Remoto Manual = True
   // e Se FALHA = False
   // } 
   // Habilita botão para ligar manualmente pela IHM.
   // Caso a bomba esteja em REMOTO e a chave foi passada para LOCAL, A bomba é  colocada em modo REMOTO MANUAL E desligada. Desse modo, ao girar  novamente de LOCAL para REMOTO, é preciso que o  operador acione manualmente para ligar a bomba ou coloque manualmente em modo REMOTO AUTOMÁTICO. Isso acontece independente do estado em que a bomba se encontrava antes de girar de REMOTO para LOCAL, garantindo assim, segurança em casos de manutenção.
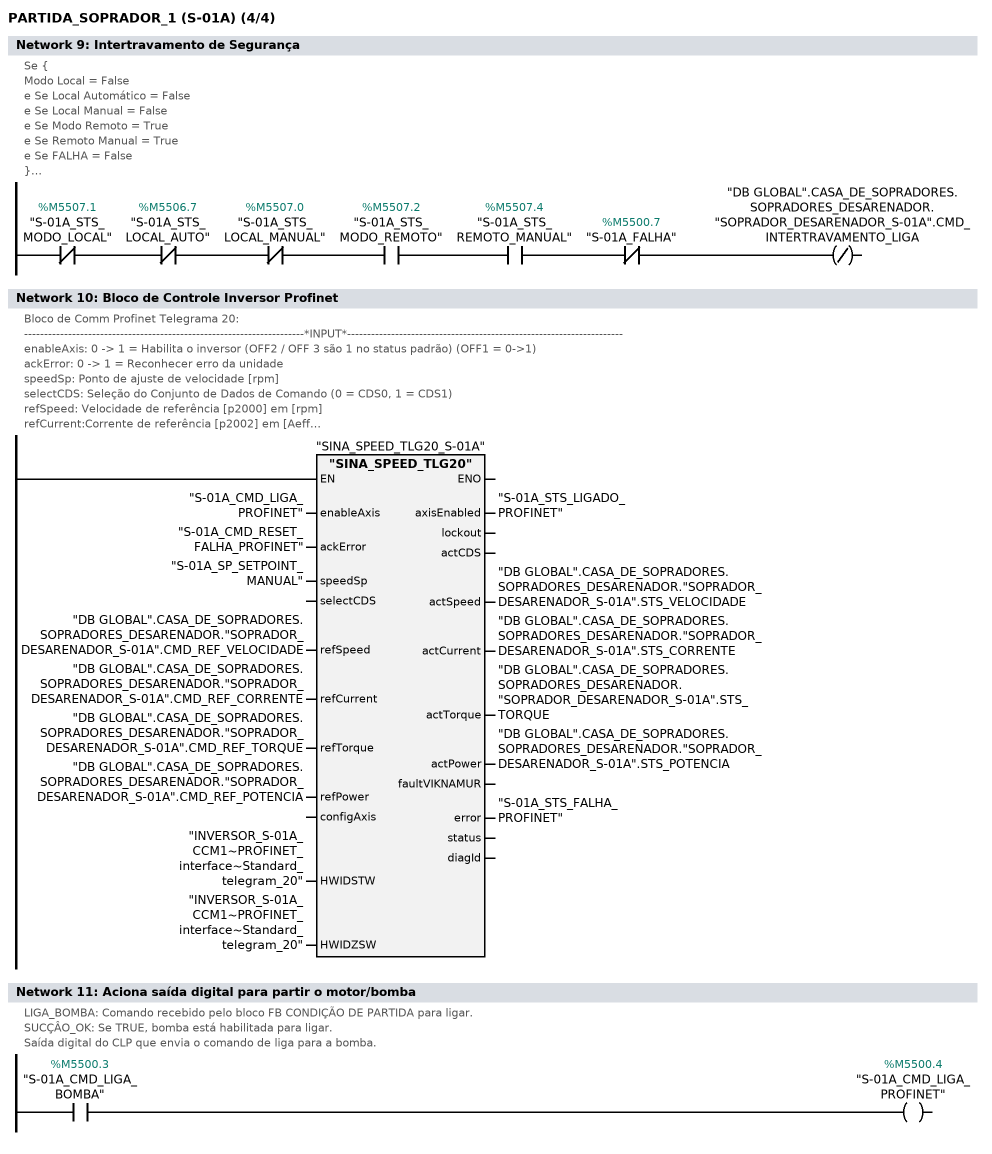
   RUNG wire#powerrail
      I_Contact( "S-01A_STS_MODO_LOCAL" )
      I_Contact( "S-01A_STS_LOCAL_AUTO" )
      I_Contact( "S-01A_STS_LOCAL_MANUAL" )
      Contact( "S-01A_STS_MODO_REMOTO" )
      Contact( "S-01A_STS_REMOTO_MANUAL" )
      I_Contact( "S-01A_FALHA" )
      I_Coil( "DB GLOBAL".CASA_DE_SOPRADORES.SOPRADORES_DESARENADOR."SOPRADOR_DESARENADOR_S-01A".CMD_INTERTRAVAMENTO_LIGA )
   END_RUNG
   // the same network as SCL:
   "DB GLOBAL".CASA_DE_SOPRADORES.SOPRADORES_DESARENADOR."SOPRADOR_DESARENADOR_S-01A".CMD_INTERTRAVAMENTO_LIGA := NOT (NOT "S-01A_STS_MODO_LOCAL" AND NOT "S-01A_STS_LOCAL_AUTO" AND NOT "S-01A_STS_LOCAL_MANUAL" AND "S-01A_STS_MODO_REMOTO" AND "S-01A_STS_REMOTO_MANUAL" AND NOT "S-01A_FALHA");
END_REGION

REGION Network 10: Bloco de Controle Inversor Profinet
   // Bloco de Comm Profinet Telegrama 20:
   // ----------------------------------------------------------------------*INPUT*---------------------------------------------------------------------
   // enableAxis: 0 -> 1 = Habilita o inversor (OFF2 / OFF 3 são 1 no status padrão) (OFF1 = 0->1)
   // ackError: 0 -> 1 = Reconhecer erro da unidade
   // speedSp: Ponto de ajuste de velocidade [rpm]
   // selectCDS: Seleção do Conjunto de Dados de Comando (0 = CDS0, 1 = CDS1)
   // refSpeed: Velocidade de referência [p2000] em [rpm]
   // refCurrent:Corrente de referência [p2002] em [Aeff]
   // refTorque: Torque de referência [p2003] em [Nm]
   // refPower: Potência de referência [r2005] em [kW]
   // configAxis: Entrada binária programada para controlar todas as funções do telegrama sem sua própria entrada de bloco de função
   // HWIDSTW: Slot de ponto de ajuste do identificador de hardware
   // HWIDZSW: Slot de valor real do identificador de hardware
   // ---------------------------------------------------------------------*OUTPUT*------------------------------------------------------------------
   // axisEnabled: 1 = O inversor está habilitado
   // lockout: 1 = Bloqueio do inversor ativo
   // actCDS: Conjunto de dados de comando ativo (0 = CDS0, 1 = CDS1)
   // actSpeed: Velocidade real suavizada em [1/min]
   // actCurrent: Corrente real suavizada em [Arms]
   // actTorque: Torque real suavizado em [Nm]
   // actPower: Potência ativa real suavizada em [kW]
   // faultVIKNAMUR: Palavra de falha de acordo com a definição VIK-NAMUR
   // error: 1 = Erro (FB e Infeed)
   // status: Saída de status (7002 = FB em operação; 7xxx = aviso; 8xxx = descrição do erro - leia o manual)
   // diagId: Códigos de erro dos blocos funcionais do sistema DPWR / DPRD_DAT
   RUNG wire#powerrail
      "SINA_SPEED_TLG20_S-01A"(enableAxis := "S-01A_CMD_LIGA_PROFINET", ackError := "S-01A_CMD_RESET_FALHA_PROFINET", speedSp := "S-01A_SP_SETPOINT_MANUAL", selectCDS :=, refSpeed := "DB GLOBAL".CASA_DE_SOPRADORES.SOPRADORES_DESARENADOR."SOPRADOR_DESARENADOR_S-01A".CMD_REF_VELOCIDADE, refCurrent := "DB GLOBAL".CASA_DE_SOPRADORES.SOPRADORES_DESARENADOR."SOPRADOR_DESARENADOR_S-01A".CMD_REF_CORRENTE, refTorque := "DB GLOBAL".CASA_DE_SOPRADORES.SOPRADORES_DESARENADOR."SOPRADOR_DESARENADOR_S-01A".CMD_REF_TORQUE, refPower := "DB GLOBAL".CASA_DE_SOPRADORES.SOPRADORES_DESARENADOR."SOPRADOR_DESARENADOR_S-01A".CMD_REF_POTENCIA, configAxis :=, HWIDSTW := "INVERSOR_S-01A_CCM1~PROFINET_interface~Standard_telegram_20", HWIDZSW := "INVERSOR_S-01A_CCM1~PROFINET_interface~Standard_telegram_20", axisEnabled => "S-01A_STS_LIGADO_PROFINET", lockout =>, actCDS =>, actSpeed => "DB GLOBAL".CASA_DE_SOPRADORES.SOPRADORES_DESARENADOR."SOPRADOR_DESARENADOR_S-01A".STS_VELOCIDADE, actCurrent => "DB GLOBAL".CASA_DE_SOPRADORES.SOPRADORES_DESARENADOR."SOPRADOR_DESARENADOR_S-01A".STS_CORRENTE, actTorque => "DB GLOBAL".CASA_DE_SOPRADORES.SOPRADORES_DESARENADOR."SOPRADOR_DESARENADOR_S-01A".STS_TORQUE, actPower => "DB GLOBAL".CASA_DE_SOPRADORES.SOPRADORES_DESARENADOR."SOPRADOR_DESARENADOR_S-01A".STS_POTENCIA, faultVIKNAMUR =>, error => "S-01A_STS_FALHA_PROFINET", status =>, diagId =>)
   END_RUNG
   // the same network as SCL:
   "SINA_SPEED_TLG20_S-01A"(enableAxis := "S-01A_CMD_LIGA_PROFINET",   // "SINA_SPEED_TLG20"
                           ackError := "S-01A_CMD_RESET_FALHA_PROFINET",
                           speedSp := "S-01A_SP_SETPOINT_MANUAL",
                           refSpeed := "DB GLOBAL".CASA_DE_SOPRADORES.SOPRADORES_DESARENADOR."SOPRADOR_DESARENADOR_S-01A".CMD_REF_VELOCIDADE,
                           refCurrent := "DB GLOBAL".CASA_DE_SOPRADORES.SOPRADORES_DESARENADOR."SOPRADOR_DESARENADOR_S-01A".CMD_REF_CORRENTE,
                           refTorque := "DB GLOBAL".CASA_DE_SOPRADORES.SOPRADORES_DESARENADOR."SOPRADOR_DESARENADOR_S-01A".CMD_REF_TORQUE,
                           refPower := "DB GLOBAL".CASA_DE_SOPRADORES.SOPRADORES_DESARENADOR."SOPRADOR_DESARENADOR_S-01A".CMD_REF_POTENCIA,
                           HWIDSTW := "INVERSOR_S-01A_CCM1~PROFINET_interface~Standard_telegram_20",
                           HWIDZSW := "INVERSOR_S-01A_CCM1~PROFINET_interface~Standard_telegram_20",
                           axisEnabled => "S-01A_STS_LIGADO_PROFINET",
                           actSpeed => "DB GLOBAL".CASA_DE_SOPRADORES.SOPRADORES_DESARENADOR."SOPRADOR_DESARENADOR_S-01A".STS_VELOCIDADE,
                           actCurrent => "DB GLOBAL".CASA_DE_SOPRADORES.SOPRADORES_DESARENADOR."SOPRADOR_DESARENADOR_S-01A".STS_CORRENTE,
                           actTorque => "DB GLOBAL".CASA_DE_SOPRADORES.SOPRADORES_DESARENADOR."SOPRADOR_DESARENADOR_S-01A".STS_TORQUE,
                           actPower => "DB GLOBAL".CASA_DE_SOPRADORES.SOPRADORES_DESARENADOR."SOPRADOR_DESARENADOR_S-01A".STS_POTENCIA,
                           error => "S-01A_STS_FALHA_PROFINET");
END_REGION

REGION Network 11: Aciona saída digital para partir o motor/bomba
   // LIGA_BOMBA: Comando recebido pelo bloco FB CONDIÇÃO DE PARTIDA para ligar.
   // SUCÇÂO_OK: Se TRUE, bomba está habilitada para ligar.
   // 
   // Saída digital do CLP que envia o comando de liga para a bomba.
   RUNG wire#powerrail
      Contact( "S-01A_CMD_LIGA_BOMBA" )
      Coil( "S-01A_CMD_LIGA_PROFINET" )
   END_RUNG
   // the same network as SCL:
   "S-01A_CMD_LIGA_PROFINET" := "S-01A_CMD_LIGA_BOMBA";
END_REGION
END_FUNCTION

FUNCTION "FC_Modelo" : Void   // FC516, LAD
TITLE = Montagem de Word de Alarmes
{ S7_Optimized_Access := 'TRUE' }
VERSION : 0.1
// stored: AutoNumber true, IsIECCheckEnabled false, SetENOAutomatically false, UDAEnableTagReadback false
BEGIN

REGION Network 1
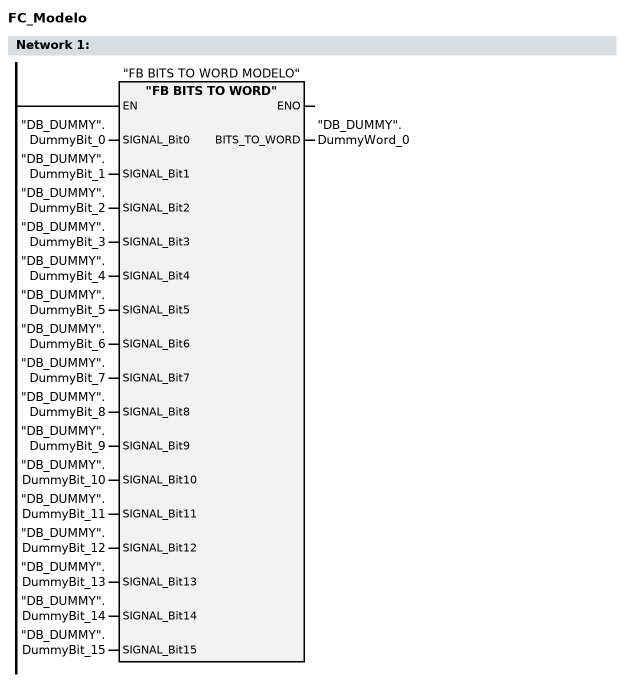
   RUNG wire#powerrail
      "FB BITS TO WORD MODELO"(SIGNAL_Bit0 := "DB_DUMMY".DummyBit_0, SIGNAL_Bit1 := "DB_DUMMY".DummyBit_1, SIGNAL_Bit2 := "DB_DUMMY".DummyBit_2, SIGNAL_Bit3 := "DB_DUMMY".DummyBit_3, SIGNAL_Bit4 := "DB_DUMMY".DummyBit_4, SIGNAL_Bit5 := "DB_DUMMY".DummyBit_5, SIGNAL_Bit6 := "DB_DUMMY".DummyBit_6, SIGNAL_Bit7 := "DB_DUMMY".DummyBit_7, SIGNAL_Bit8 := "DB_DUMMY".DummyBit_8, SIGNAL_Bit9 := "DB_DUMMY".DummyBit_9, SIGNAL_Bit10 := "DB_DUMMY".DummyBit_10, SIGNAL_Bit11 := "DB_DUMMY".DummyBit_11, SIGNAL_Bit12 := "DB_DUMMY".DummyBit_12, SIGNAL_Bit13 := "DB_DUMMY".DummyBit_13, SIGNAL_Bit14 := "DB_DUMMY".DummyBit_14, SIGNAL_Bit15 := "DB_DUMMY".DummyBit_15, BITS_TO_WORD => "DB_DUMMY".DummyWord_0)
   END_RUNG
   // the same network as SCL:
   "FB BITS TO WORD MODELO"(SIGNAL_Bit0 := "DB_DUMMY".DummyBit_0,   // "FB BITS TO WORD"
                           SIGNAL_Bit1 := "DB_DUMMY".DummyBit_1,
                           SIGNAL_Bit2 := "DB_DUMMY".DummyBit_2,
                           SIGNAL_Bit3 := "DB_DUMMY".DummyBit_3,
                           SIGNAL_Bit4 := "DB_DUMMY".DummyBit_4,
                           SIGNAL_Bit5 := "DB_DUMMY".DummyBit_5,
                           SIGNAL_Bit6 := "DB_DUMMY".DummyBit_6,
                           SIGNAL_Bit7 := "DB_DUMMY".DummyBit_7,
                           SIGNAL_Bit8 := "DB_DUMMY".DummyBit_8,
                           SIGNAL_Bit9 := "DB_DUMMY".DummyBit_9,
                           SIGNAL_Bit10 := "DB_DUMMY".DummyBit_10,
                           SIGNAL_Bit11 := "DB_DUMMY".DummyBit_11,
                           SIGNAL_Bit12 := "DB_DUMMY".DummyBit_12,
                           SIGNAL_Bit13 := "DB_DUMMY".DummyBit_13,
                           SIGNAL_Bit14 := "DB_DUMMY".DummyBit_14,
                           SIGNAL_Bit15 := "DB_DUMMY".DummyBit_15,
                           BITS_TO_WORD => "DB_DUMMY".DummyWord_0);
END_REGION
END_FUNCTION

FUNCTION_BLOCK "FB BITS TO WORD"
{ S7_Optimized_Access := 'TRUE' }
VERSION : 0.1
VAR_INPUT
   SIGNAL_Bit0 : Bool;
   SIGNAL_Bit1 : Bool;
   SIGNAL_Bit2 : Bool;
   SIGNAL_Bit3 : Bool;
   SIGNAL_Bit4 : Bool;
   SIGNAL_Bit5 : Bool;
   SIGNAL_Bit6 : Bool;
   SIGNAL_Bit7 : Bool;
   SIGNAL_Bit8 : Bool;
   SIGNAL_Bit9 : Bool;
   SIGNAL_Bit10 : Bool;
   SIGNAL_Bit11 : Bool;
   SIGNAL_Bit12 : Bool;
   SIGNAL_Bit13 : Bool;
   SIGNAL_Bit14 : Bool;
   SIGNAL_Bit15 : Bool;
END_VAR
VAR_OUTPUT
   BITS_TO_WORD : Word;
END_VAR

BEGIN
   BITS_TO_WORD.%X0 := #SIGNAL_Bit0;
   BITS_TO_WORD.%X1 := #SIGNAL_Bit1;
   BITS_TO_WORD.%X2 := #SIGNAL_Bit2;
   BITS_TO_WORD.%X3 := #SIGNAL_Bit3;
   BITS_TO_WORD.%X4 := #SIGNAL_Bit4;
   BITS_TO_WORD.%X5 := #SIGNAL_Bit5;
   BITS_TO_WORD.%X6 := #SIGNAL_Bit6;
   BITS_TO_WORD.%X7 := #SIGNAL_Bit7;
   BITS_TO_WORD.%X8 := #SIGNAL_Bit8;
   BITS_TO_WORD.%X9 := #SIGNAL_Bit9;
   BITS_TO_WORD.%X10 := #SIGNAL_Bit10;
   BITS_TO_WORD.%X11 := #SIGNAL_Bit11;
   BITS_TO_WORD.%X12 := #SIGNAL_Bit12;
   BITS_TO_WORD.%X13 := #SIGNAL_Bit13;
   BITS_TO_WORD.%X14 := #SIGNAL_Bit14;
   BITS_TO_WORD.%X15 := #SIGNAL_Bit15;
END_FUNCTION_BLOCK

DATA_BLOCK "DB_BITS_TO_WORD_MODELO"
{ S7_Optimized_Access := 'TRUE' }
VERSION : 0.1
"FB BITS TO WORD"

BEGIN
END_DATA_BLOCK

DATA_BLOCK "DB GLOBAL"
{ S7_Optimized_Access := 'TRUE' }
VERSION : 0.1
   STRUCT
      "Motor_BH-01A" : "MotorDados";
      "Motor_BH-01B" : "MotorDados";
      ETA : STRUCT
         ALARMES : STRUCT
            WORD_ALARMES_1 : Word;
            WORD_ALARMES_2 : Word;
         END_STRUCT;
      END_STRUCT;
   END_STRUCT;

BEGIN
END_DATA_BLOCK

FUNCTION "MOLDE_ANALOGS" : Void   // FC128, LAD
{ S7_Optimized_Access := 'TRUE' }
VERSION : 0.1
// Parâmetros da Equação da Reta
// ANALOG_IN_4a20mA: Entrada Analógica
// Y1_CONFIG: Range mínimo Sinal de Campo
// Y2_CONFIG: Range máximo Sinal de Campo
// X1_CONFIG: Range Mínimo Entrada Analógica CLP
// X2_CONFIG: Range Máximo Entrada Analógica CLP
// COMANDO: Parâmetro enviado da IHM/SCADA
// COMANDO_VALOR: Parâmetro referente à aferição do bloco
// GRANDEZA_MAX = Valor de comunicação RS485, enviado pelo inversor 
// RANGE_MIN_CADASTRADO = Valor de leitura minimo que irá aparecer no display IHM
// RANGE_MAX_CADASTRADO = Valor de leitura maximo que irá aparecer no display IHM
// 
// Comando Aferição 8888: (FQIT-01)
// Comando Limites 9999: (FQIT-01)
// stored: AutoNumber true, IsIECCheckEnabled false, SetENOAutomatically false, UDAEnableTagReadback false
BEGIN

REGION Network 1: Aferição Equipamento (FQIT-01)
   // Aferição Entrada Analógica (FQIT-01)
   // 
   // Comando:
   // 8888: Comando de Aferição (FQIT-01)
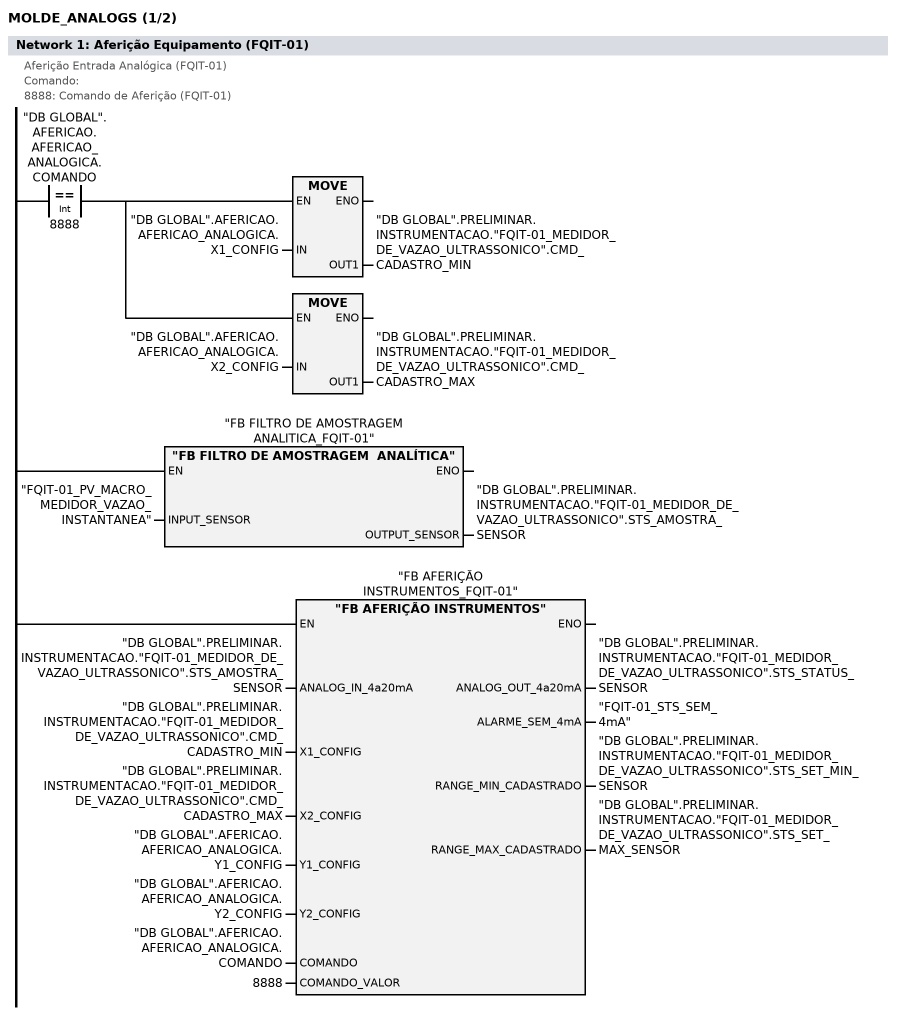
   RUNG wire#powerrail
      { S7_Templates := "SrcType := Int" } EQ_Contact(in1 := "DB GLOBAL".AFERICAO.AFERICAO_ANALOGICA.COMANDO, in2 := 8888)
      wire#w1
      Move(in := "DB GLOBAL".AFERICAO.AFERICAO_ANALOGICA.X1_CONFIG, out1 => "DB GLOBAL".PRELIMINAR.INSTRUMENTACAO."FQIT-01_MEDIDOR_DE_VAZAO_ULTRASSONICO".CMD_CADASTRO_MIN)
   END_RUNG
   RUNG wire#w1
      Move(in := "DB GLOBAL".AFERICAO.AFERICAO_ANALOGICA.X2_CONFIG, out1 => "DB GLOBAL".PRELIMINAR.INSTRUMENTACAO."FQIT-01_MEDIDOR_DE_VAZAO_ULTRASSONICO".CMD_CADASTRO_MAX)
   END_RUNG
   RUNG wire#powerrail
      "FB FILTRO DE AMOSTRAGEM  ANALITICA_FQIT-01"(INPUT_SENSOR := "FQIT-01_PV_MACRO_MEDIDOR_VAZAO_INSTANTANEA", OUTPUT_SENSOR => "DB GLOBAL".PRELIMINAR.INSTRUMENTACAO."FQIT-01_MEDIDOR_DE_VAZAO_ULTRASSONICO".STS_AMOSTRA_SENSOR)
   END_RUNG
   RUNG wire#powerrail
      "FB AFERIÇÃO INSTRUMENTOS_FQIT-01"(ANALOG_IN_4a20mA := "DB GLOBAL".PRELIMINAR.INSTRUMENTACAO."FQIT-01_MEDIDOR_DE_VAZAO_ULTRASSONICO".STS_AMOSTRA_SENSOR, X1_CONFIG := "DB GLOBAL".PRELIMINAR.INSTRUMENTACAO."FQIT-01_MEDIDOR_DE_VAZAO_ULTRASSONICO".CMD_CADASTRO_MIN, X2_CONFIG := "DB GLOBAL".PRELIMINAR.INSTRUMENTACAO."FQIT-01_MEDIDOR_DE_VAZAO_ULTRASSONICO".CMD_CADASTRO_MAX, Y1_CONFIG := "DB GLOBAL".AFERICAO.AFERICAO_ANALOGICA.Y1_CONFIG, Y2_CONFIG := "DB GLOBAL".AFERICAO.AFERICAO_ANALOGICA.Y2_CONFIG, COMANDO := "DB GLOBAL".AFERICAO.AFERICAO_ANALOGICA.COMANDO, COMANDO_VALOR := 8888, ANALOG_OUT_4a20mA => "DB GLOBAL".PRELIMINAR.INSTRUMENTACAO."FQIT-01_MEDIDOR_DE_VAZAO_ULTRASSONICO".STS_STATUS_SENSOR, ALARME_SEM_4mA => "FQIT-01_STS_SEM_4mA", RANGE_MIN_CADASTRADO => "DB GLOBAL".PRELIMINAR.INSTRUMENTACAO."FQIT-01_MEDIDOR_DE_VAZAO_ULTRASSONICO".STS_SET_MIN_SENSOR, RANGE_MAX_CADASTRADO => "DB GLOBAL".PRELIMINAR.INSTRUMENTACAO."FQIT-01_MEDIDOR_DE_VAZAO_ULTRASSONICO".STS_SET_MAX_SENSOR)
   END_RUNG
   // the same network as SCL:
   IF "DB GLOBAL".AFERICAO.AFERICAO_ANALOGICA.COMANDO = 8888 THEN
       "DB GLOBAL".PRELIMINAR.INSTRUMENTACAO."FQIT-01_MEDIDOR_DE_VAZAO_ULTRASSONICO".CMD_CADASTRO_MIN := "DB GLOBAL".AFERICAO.AFERICAO_ANALOGICA.X1_CONFIG;
       "DB GLOBAL".PRELIMINAR.INSTRUMENTACAO."FQIT-01_MEDIDOR_DE_VAZAO_ULTRASSONICO".CMD_CADASTRO_MAX := "DB GLOBAL".AFERICAO.AFERICAO_ANALOGICA.X2_CONFIG;
   END_IF;
   "FB FILTRO DE AMOSTRAGEM  ANALITICA_FQIT-01"(INPUT_SENSOR := "FQIT-01_PV_MACRO_MEDIDOR_VAZAO_INSTANTANEA",   // "FB FILTRO DE AMOSTRAGEM  ANALÍTICA"
                           OUTPUT_SENSOR => "DB GLOBAL".PRELIMINAR.INSTRUMENTACAO."FQIT-01_MEDIDOR_DE_VAZAO_ULTRASSONICO".STS_AMOSTRA_SENSOR);
   "FB AFERIÇÃO INSTRUMENTOS_FQIT-01"(ANALOG_IN_4a20mA := "DB GLOBAL".PRELIMINAR.INSTRUMENTACAO."FQIT-01_MEDIDOR_DE_VAZAO_ULTRASSONICO".STS_AMOSTRA_SENSOR,   // "FB AFERIÇÃO INSTRUMENTOS"
                           X1_CONFIG := "DB GLOBAL".PRELIMINAR.INSTRUMENTACAO."FQIT-01_MEDIDOR_DE_VAZAO_ULTRASSONICO".CMD_CADASTRO_MIN,
                           X2_CONFIG := "DB GLOBAL".PRELIMINAR.INSTRUMENTACAO."FQIT-01_MEDIDOR_DE_VAZAO_ULTRASSONICO".CMD_CADASTRO_MAX,
                           Y1_CONFIG := "DB GLOBAL".AFERICAO.AFERICAO_ANALOGICA.Y1_CONFIG,
                           Y2_CONFIG := "DB GLOBAL".AFERICAO.AFERICAO_ANALOGICA.Y2_CONFIG,
                           COMANDO := "DB GLOBAL".AFERICAO.AFERICAO_ANALOGICA.COMANDO,
                           COMANDO_VALOR := 8888,
                           ANALOG_OUT_4a20mA => "DB GLOBAL".PRELIMINAR.INSTRUMENTACAO."FQIT-01_MEDIDOR_DE_VAZAO_ULTRASSONICO".STS_STATUS_SENSOR,
                           ALARME_SEM_4mA => "FQIT-01_STS_SEM_4mA",
                           RANGE_MIN_CADASTRADO => "DB GLOBAL".PRELIMINAR.INSTRUMENTACAO."FQIT-01_MEDIDOR_DE_VAZAO_ULTRASSONICO".STS_SET_MIN_SENSOR,
                           RANGE_MAX_CADASTRADO => "DB GLOBAL".PRELIMINAR.INSTRUMENTACAO."FQIT-01_MEDIDOR_DE_VAZAO_ULTRASSONICO".STS_SET_MAX_SENSOR);
END_REGION

REGION Network 2: Limites de Operação (FQIT-01)
   // Cadastro Limites de Operação sensor (FQIT-01)
   // Alarme leitura muito baixa
   // Alarme leitura baixa
   // Alarme leitura alta
   // Alarme leitura muito alta
   // 
   // Comando:
   // 9999: Definição de Limites para (FQIT-01)
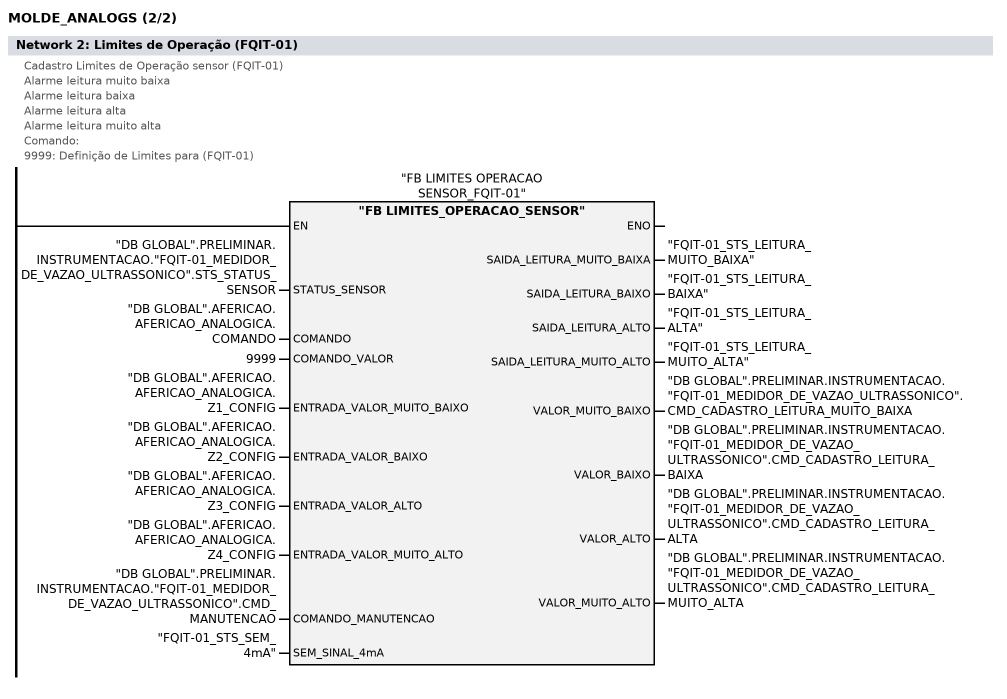
   RUNG wire#powerrail
      "FB LIMITES OPERACAO SENSOR_FQIT-01"(STATUS_SENSOR := "DB GLOBAL".PRELIMINAR.INSTRUMENTACAO."FQIT-01_MEDIDOR_DE_VAZAO_ULTRASSONICO".STS_STATUS_SENSOR, COMANDO := "DB GLOBAL".AFERICAO.AFERICAO_ANALOGICA.COMANDO, COMANDO_VALOR := 9999, ENTRADA_VALOR_MUITO_BAIXO := "DB GLOBAL".AFERICAO.AFERICAO_ANALOGICA.Z1_CONFIG, ENTRADA_VALOR_BAIXO := "DB GLOBAL".AFERICAO.AFERICAO_ANALOGICA.Z2_CONFIG, ENTRADA_VALOR_ALTO := "DB GLOBAL".AFERICAO.AFERICAO_ANALOGICA.Z3_CONFIG, ENTRADA_VALOR_MUITO_ALTO := "DB GLOBAL".AFERICAO.AFERICAO_ANALOGICA.Z4_CONFIG, COMANDO_MANUTENCAO := "DB GLOBAL".PRELIMINAR.INSTRUMENTACAO."FQIT-01_MEDIDOR_DE_VAZAO_ULTRASSONICO".CMD_MANUTENCAO, SEM_SINAL_4mA := "FQIT-01_STS_SEM_4mA", SAIDA_LEITURA_MUITO_BAIXA => "FQIT-01_STS_LEITURA_MUITO_BAIXA", SAIDA_LEITURA_BAIXO => "FQIT-01_STS_LEITURA_BAIXA", SAIDA_LEITURA_ALTO => "FQIT-01_STS_LEITURA_ALTA", SAIDA_LEITURA_MUITO_ALTO => "FQIT-01_STS_LEITURA_MUITO_ALTA", VALOR_MUITO_BAIXO => "DB GLOBAL".PRELIMINAR.INSTRUMENTACAO."FQIT-01_MEDIDOR_DE_VAZAO_ULTRASSONICO".CMD_CADASTRO_LEITURA_MUITO_BAIXA, VALOR_BAIXO => "DB GLOBAL".PRELIMINAR.INSTRUMENTACAO."FQIT-01_MEDIDOR_DE_VAZAO_ULTRASSONICO".CMD_CADASTRO_LEITURA_BAIXA, VALOR_ALTO => "DB GLOBAL".PRELIMINAR.INSTRUMENTACAO."FQIT-01_MEDIDOR_DE_VAZAO_ULTRASSONICO".CMD_CADASTRO_LEITURA_ALTA, VALOR_MUITO_ALTO => "DB GLOBAL".PRELIMINAR.INSTRUMENTACAO."FQIT-01_MEDIDOR_DE_VAZAO_ULTRASSONICO".CMD_CADASTRO_LEITURA_MUITO_ALTA)
   END_RUNG
   // the same network as SCL:
   "FB LIMITES OPERACAO SENSOR_FQIT-01"(STATUS_SENSOR := "DB GLOBAL".PRELIMINAR.INSTRUMENTACAO."FQIT-01_MEDIDOR_DE_VAZAO_ULTRASSONICO".STS_STATUS_SENSOR,   // "FB LIMITES_OPERACAO_SENSOR"
                           COMANDO := "DB GLOBAL".AFERICAO.AFERICAO_ANALOGICA.COMANDO,
                           COMANDO_VALOR := 9999,
                           ENTRADA_VALOR_MUITO_BAIXO := "DB GLOBAL".AFERICAO.AFERICAO_ANALOGICA.Z1_CONFIG,
                           ENTRADA_VALOR_BAIXO := "DB GLOBAL".AFERICAO.AFERICAO_ANALOGICA.Z2_CONFIG,
                           ENTRADA_VALOR_ALTO := "DB GLOBAL".AFERICAO.AFERICAO_ANALOGICA.Z3_CONFIG,
                           ENTRADA_VALOR_MUITO_ALTO := "DB GLOBAL".AFERICAO.AFERICAO_ANALOGICA.Z4_CONFIG,
                           COMANDO_MANUTENCAO := "DB GLOBAL".PRELIMINAR.INSTRUMENTACAO."FQIT-01_MEDIDOR_DE_VAZAO_ULTRASSONICO".CMD_MANUTENCAO,
                           SEM_SINAL_4mA := "FQIT-01_STS_SEM_4mA",
                           SAIDA_LEITURA_MUITO_BAIXA => "FQIT-01_STS_LEITURA_MUITO_BAIXA",
                           SAIDA_LEITURA_BAIXO => "FQIT-01_STS_LEITURA_BAIXA",
                           SAIDA_LEITURA_ALTO => "FQIT-01_STS_LEITURA_ALTA",
                           SAIDA_LEITURA_MUITO_ALTO => "FQIT-01_STS_LEITURA_MUITO_ALTA",
                           VALOR_MUITO_BAIXO => "DB GLOBAL".PRELIMINAR.INSTRUMENTACAO."FQIT-01_MEDIDOR_DE_VAZAO_ULTRASSONICO".CMD_CADASTRO_LEITURA_MUITO_BAIXA,
                           VALOR_BAIXO => "DB GLOBAL".PRELIMINAR.INSTRUMENTACAO."FQIT-01_MEDIDOR_DE_VAZAO_ULTRASSONICO".CMD_CADASTRO_LEITURA_BAIXA,
                           VALOR_ALTO => "DB GLOBAL".PRELIMINAR.INSTRUMENTACAO."FQIT-01_MEDIDOR_DE_VAZAO_ULTRASSONICO".CMD_CADASTRO_LEITURA_ALTA,
                           VALOR_MUITO_ALTO => "DB GLOBAL".PRELIMINAR.INSTRUMENTACAO."FQIT-01_MEDIDOR_DE_VAZAO_ULTRASSONICO".CMD_CADASTRO_LEITURA_MUITO_ALTA);
END_REGION
END_FUNCTION

FUNCTION "FC_SmokeSrc" : Void
{ S7_Optimized_Access := 'TRUE' }
VERSION : 0.1
BEGIN
    IF "Smoke_Bit" THEN
        "Smoke_Int" := 42;
    END_IF;
END_FUNCTION

FUNCTION "FC_Example" : Void
{ S7_Optimized_Access := 'TRUE' }
VERSION : 0.1
   VAR_INPUT
      iEnable : Bool;
   END_VAR
   VAR_OUTPUT
      qActive : Bool;
   END_VAR

BEGIN
    #qActive := #iEnable;
END_FUNCTION

FUNCTION_BLOCK "ZZ_TESTE_SCL"
{ S7_Optimized_Access := 'TRUE' }
VERSION : 0.1
   VAR_INPUT
      RUN : Bool;
      RAW : Int;
   END_VAR
   VAR_OUTPUT
      DONE : Bool;
      ENG : Real;
   END_VAR
   VAR
      TIMER_ON : TON_TIME;
   END_VAR

BEGIN
    #TIMER_ON(IN := #RUN, PT := T#5S);
    #DONE := #TIMER_ON.Q;
    #ENG := SCALE_X(MIN := 0.0, VALUE := NORM_X(MIN := 0, VALUE := #RAW, MAX := 27648), MAX := 100.0);
END_FUNCTION_BLOCK

FUNCTION "FC_LadderDemo" : Void
// Subset aceito por: tia import-ladder --file ladder.scl
// Só tags globais (com ou sem aspas). Sem #locais, FOR/WHILE/CASE, aritmética.
BEGIN
    // Rede 1 — selo com série/paralelo
    "Cmd_Motor1" := ("Start" OR "Cmd_Motor1") AND NOT "Stop" AND NOT "Falha_M1";

    // Rede 2 — Set
    IF "Nivel_Alto" AND "Auto" THEN "Alarme" := TRUE; END_IF;

    // Rede 3 — Reset
    IF "Reset" THEN "Alarme" := FALSE; END_IF;

    // Rede 4 — coil simples via IF/ELSE
    IF "Auto" AND NOT "Manutencao" THEN "Pronto" := TRUE; ELSE "Pronto" := FALSE; END_IF;

    // Rede 5 — comparador como contato
    "Temp_OK" := "Temperatura" > 50 AND NOT "Sensor_Falha";

    // Rede 6 — MOVE condicional de literal
    IF "Auto" THEN "Setpoint" := 75; END_IF;
END_FUNCTION
